Yaskawa INFORM job: R2_W27-A2(70,-90)_MP_OK.JBI

/JOB
//NAME R2_W27-A2(70,-90)_MP_OK
///FOLDERNAME MP_TEST
//POS
///NPOS 130,130,0,4,0,0
///TOOL 0
///POSTYPE PULSE
///PULSE
C00000=102318,51059,-6827,-6506,109190,54954
C00001=121032,58356,65608,-5376,86027,77236
C00002=120656,64598,75406,-5436,83192,77232
C00003=120505,64053,76314,-5460,82347,77219
C00004=120511,67645,82265,-5481,80539,77299
C00005=120505,64053,76314,-5460,82347,77219
C00006=120199,65070,76942,-5493,82463,77112
C00007=120032,61399,73230,-5508,82846,77040
C00008=120199,65070,76942,-5493,82463,77112
C00009=121567,62706,73730,-5333,83311,77530
C00010=121293,57658,68714,-5360,83784,77419
C00011=120253,58213,69266,-5476,83660,77079
C00012=121293,57658,68714,-5360,83784,77419
C00013=121567,62706,73730,-5333,83311,77530
C00014=120505,64053,76314,-5460,82347,77219
C00015=120656,64598,75406,-5436,83192,77232
C00016=121032,58526,65774,-5376,86013,77236
C00017=93357,59983,67350,2576,87301,77052
C00018=93973,65449,76277,2662,84599,77201
C00019=93950,64770,77022,2661,83793,77176
C00020=94041,68208,82724,2681,82050,77169
C00021=93950,64770,77022,2661,83793,77176
C00022=94821,64601,76206,2774,84179,77472
C00023=94634,60689,72295,2749,84583,77418
C00024=94821,64601,76206,2774,84179,77472
C00025=93392,64700,76725,2587,83958,76996
C00026=93160,58385,69524,2553,85150,76943
C00027=94147,57298,68173,2682,85392,77275
C00028=93160,58385,69524,2553,85150,76943
C00029=93392,64700,76725,2587,83958,76996
C00030=93950,64770,77022,2661,83793,77176
C00031=93973,65449,76277,2662,84599,77201
C00032=93336,59773,67146,2573,87319,77046
C00033=95545,69101,76731,-2374,84009,73270
C00034=95160,67852,79145,-2422,81872,73183
C00035=95003,67493,80298,-2443,80974,73148
C00036=94849,62700,75029,-2455,81748,73082
C00037=95003,67493,80298,-2443,80974,73148
C00038=93105,70422,84610,-2644,79768,72546
C00039=92524,67765,81382,-2700,80371,72342
C00040=93361,68913,82672,-2615,80194,72622
C00041=94751,59758,68035,-2453,84535,72995
C00042=92805,53349,62303,-2649,84709,72342
C00043=92901,55574,66096,-2644,83522,72399
C00044=92805,53349,62303,-2649,84709,72342
C00045=94751,59758,68035,-2453,84535,72995
C00046=95003,67493,80298,-2443,80974,73148
C00047=95160,67852,79145,-2422,81872,73183
C00048=95545,69101,76731,-2374,84009,73270
C00049=107317,62571,74358,10654,88778,76029
C00050=107317,56363,61014,10704,93717,76452
C00051=107317,62472,74242,10653,88798,76031
C00052=107230,62000,74261,10636,88556,75982
C00053=107581,65118,76915,10703,88484,76092
C00054=107323,60406,70480,10660,90030,76138
C00055=107264,61783,74050,10643,88577,75994
C00056=107253,61475,73709,10642,88626,75994
C00057=107117,62576,75125,9124,76631,64990
C00058=107127,63032,75625,10605,72549,55451
C00059=107164,62402,74962,9975,72602,48239
C00060=107192,61809,74312,8045,73320,42963
C00061=107223,63525,76074,7091,73334,41100
C00062=107292,63418,75963,5949,73527,39196
C00063=107230,61705,73943,5940,73892,39194
C00064=107323,62660,74463,4678,74173,37311
C00065=107324,62694,74502,4678,74166,37311
C00066=107665,73796,87925,4736,71600,37329
C00067=120729,48613,37887,-12949,101575,-14829
C00068=120728,62727,74542,-12584,86628,-80773
C00069=120664,61680,73824,-12594,86525,-80783
C00070=120693,60658,70774,-12585,87849,-80908
C00071=120585,65581,77469,-12610,86279,-80786
C00072=120690,61906,74287,-12590,86368,-80759
C00073=120903,61800,74113,-12557,86448,-80696
C00074=120945,62548,75100,-8817,74987,-69882
C00075=120948,62197,74655,-9458,70881,-60435
C00076=120932,61569,73990,-8829,71047,-53224
C00077=120988,63466,76076,-6164,72080,-46036
C00078=121112,63464,75917,-5072,72564,-44073
C00079=121088,62388,74845,-3850,73000,-42173
C00080=120728,62552,74336,-3837,73380,-42308
C00081=120720,61560,72154,180,93079,81636
C00082=120721,62738,74555,180,92207,81635
C00083=120791,87813,92293,81,108616,81679
C00084=120002,63379,75221,11,92127,81398
C00085=121441,63308,75123,350,92148,81873
C00086=120870,108608,123515,114,99903,81701
C00087=120721,62723,74537,180,92210,81635
C00088=120720,62741,74558,180,92206,81635
C00089=93952,63192,75095,14290,85903,-74473
C00090=93948,63106,74994,14289,85921,-74472
C00091=93949,63106,74994,14289,85921,-74472
C00092=93949,63106,74994,14289,85921,-74472
C00093=93511,61763,72320,14213,86923,-74505
C00094=94061,66569,78930,14314,85278,-74508
C00095=93933,62856,74699,14286,85975,-74471
C00096=93933,62856,74699,14286,85975,-74471
C00097=93932,62855,74699,14286,85976,-74471
C00098=93936,62941,74800,14287,85957,-74472
C00099=93954,63189,75092,-4074,77084,-70207
C00100=93950,63103,74990,-4074,77102,-70209
C00101=93950,63090,74975,-4074,77104,-70209
C00102=93949,63085,74969,-4074,77106,-70209
C00103=94045,66011,77989,-4076,76757,-70165
C00104=93880,61095,71289,-4060,78342,-70273
C00105=93963,63270,75188,-4074,77067,-70203
C00106=93963,63275,75194,-4074,77066,-70203
C00107=93963,63288,75209,-4074,77063,-70203
C00108=93967,63374,75311,-4074,77045,-70201
C00109=93937,63000,74869,-16709,69815,76001
C00110=93934,62914,74768,-16707,69832,75997
C00111=93932,62884,74733,-16706,69838,75996
C00112=93931,62873,74719,-16706,69840,75995
C00113=94312,65792,77997,-16780,69420,76194
C00114=94250,60204,70492,-16607,71084,75933
C00115=93941,62972,74836,-16709,69822,76001
C00116=93942,62984,74850,-16709,69819,76002
C00117=93943,63013,74885,-16710,69814,76003
C00118=93947,63099,74986,-16712,69797,76007
C00119=93938,62981,74847,-7114,69680,67691
C00120=93935,62895,74746,-7113,69698,67689
C00121=93933,62866,74712,-7113,69704,67688
C00122=93933,62855,74698,-7112,69706,67688
C00123=93919,60777,70917,-7059,70955,67609
C00124=94303,65238,77063,-7147,69509,67829
C00125=93920,62687,74500,-7110,69740,67681
C00126=93920,62698,74513,-7110,69738,67682
C00127=93922,62727,74547,-7111,69732,67682
C00128=93926,62812,74648,-7112,69715,67685
C00129=51349,-6233,-27963,187,103874,81653
BC00000=194563,177624,868736
BC00001=225604,138849,769169
BC00002=225604,138849,769169
BC00003=225604,138849,769169
BC00004=225604,138849,769169
BC00005=225604,138849,769169
BC00006=225604,138849,769169
BC00007=225604,138849,769169
BC00008=225604,138849,769169
BC00009=225604,138849,769169
BC00010=225604,138849,769169
BC00011=225604,138849,769169
BC00012=225604,138849,769169
BC00013=225604,138849,769169
BC00014=225604,138849,769169
BC00015=225604,138849,769169
BC00016=225604,138849,769169
BC00017=124341,124762,768464
BC00018=124341,124762,768464
BC00019=124341,124762,768464
BC00020=124341,124762,768464
BC00021=124341,124762,768464
BC00022=124341,124762,768464
BC00023=124341,124762,768464
BC00024=124341,124762,768464
BC00025=124341,124762,768464
BC00026=124341,124762,768464
BC00027=124341,124762,768464
BC00028=124341,124762,768464
BC00029=124341,124762,768464
BC00030=124341,124762,768464
BC00031=124341,124762,768464
BC00032=124341,124762,768464
BC00033=131551,156203,1070987
BC00034=131551,156203,1070987
BC00035=131551,156203,1070987
BC00036=131551,156203,1070987
BC00037=131551,156203,1070987
BC00038=131551,156203,1070987
BC00039=131551,156203,1070987
BC00040=131551,156203,1070987
BC00041=131551,156203,1070987
BC00042=131551,156203,1070987
BC00043=131551,156203,1070987
BC00044=131551,156203,1070987
BC00045=131551,156203,1070987
BC00046=131551,156203,1070987
BC00047=131551,156203,1070987
BC00048=131551,156203,1070987
BC00049=225137,131323,879040
BC00050=223667,125139,756323
BC00051=223667,125139,756323
BC00052=223075,126867,747658
BC00053=223075,126867,747658
BC00054=223075,126867,747658
BC00055=218396,127755,746641
BC00056=215210,128375,745961
BC00057=203609,151152,766146
BC00058=201855,161532,767450
BC00059=199281,163395,767937
BC00060=195364,163337,768565
BC00061=193166,166495,764643
BC00062=190579,170342,759829
BC00063=190579,170342,759829
BC00064=187290,170589,769799
BC00065=184872,170576,795413
BC00066=184861,181079,896469
BC00067=167411,129445,757678
BC00068=167411,129445,757678
BC00069=167997,131165,748991
BC00070=167997,131165,748991
BC00071=167997,131165,748991
BC00072=172685,131992,747792
BC00073=175877,132570,746989
BC00074=187923,154884,766916
BC00075=189976,165022,768336
BC00076=192744,166728,768846
BC00077=199094,169671,765390
BC00078=201778,173472,760485
BC00079=204162,173688,760124
BC00080=205164,173670,770332
BC00081=217813,145490,1075175
BC00082=217813,150433,1060626
BC00083=217813,152410,925547
BC00084=217813,152410,1052396
BC00085=217813,152410,1052396
BC00086=217813,152407,927156
BC00087=217772,148655,1043478
BC00088=217771,143712,1064054
BC00089=114600,133818,976434
BC00090=114611,123316,875378
BC00091=110715,126262,854320
BC00092=109157,127441,845897
BC00093=109157,127441,845897
BC00094=109157,127441,845897
BC00095=146537,130921,755729
BC00096=148095,129743,764153
BC00097=151990,126796,785211
BC00098=151980,137299,886266
BC00099=101051,138319,898903
BC00100=101062,127816,797847
BC00101=99318,130341,773149
BC00102=98620,131350,763270
BC00103=98620,131350,763270
BC00104=98620,131350,763270
BC00105=60690,124587,772909
BC00106=61388,123578,782788
BC00107=63132,121053,807486
BC00108=63122,131556,908542
BC00109=157999,142083,988332
BC00110=158010,131580,887276
BC00111=159966,134490,863290
BC00112=160748,135654,853695
BC00113=160748,135654,853695
BC00114=160748,135654,853695
BC00115=123117,139629,764979
BC00116=122335,138464,774574
BC00117=120379,135554,798560
BC00118=120368,146057,899616
BC00119=145080,148155,895629
BC00120=145090,137652,794573
BC00121=146786,140154,769808
BC00122=147464,141155,759903
BC00123=147464,141155,759903
BC00124=147464,141155,759903
BC00125=185325,133893,768075
BC00126=184646,132892,777981
BC00127=182951,130390,802745
BC00128=182941,140893,903801
BC00129=217772,217062,1064053
///POSTYPE BASE
///RECTAN
///RCONF 0,0,0,0,0,0,0,0,0,0,0,0,0,0,0,0,0,0,0,0,0,0,0,0
P00006=0.222,-3.123,-1.508,0.0000,0.0000,0.0000
P00011=-2.329,-0.061,-0.282,0.0000,0.0000,0.0000
P00012=-0.183,-1.308,1.069,0.0000,0.0000,0.0000
P00013=-0.119,0.591,-2.131,0.0000,0.0000,0.0000
//INST
///DATE 2023/11/16 10:47
///ATTR SC,RW
///GROUP1 RB1,BS1
NOP
'r2_W27-A2(70,-90)
'
'Path S829
SFTOF
MOVJ C00000 BC00000 VJ=20.00
MOVJ C00001 BC00001 VJ=20.00
MOVL C00002 BC00002 V=100.0
MOVL C00003 BC00003 V=60.0
REFP 3 C00004 BC00004
CALL JOB:SEARCH-R1
SET P011 P006
SFTON P011
MOVL C00005 BC00005 V=60.0
MOVL C00006 BC00006 V=60.0
REFP 3 C00007 BC00007
CALL JOB:SEARCH-R1
SET P011 P006
SFTON P011
MOVL C00008 BC00008 V=60.0
MOVL C00009 BC00009 V=100.0
MOVL C00010 BC00010 V=60.0
REFP 3 C00011 BC00011
CALL JOB:SEARCH-R1
SET P011 P006
SFTON P011
MOVL C00012 BC00012 V=60.0
MOVL C00013 BC00013 V=100.0
MOVL C00014 BC00014 V=100.0
MOVL C00015 BC00015 V=100.0
MOVL C00016 BC00016 V=100.0
'Path S830
SFTOF
MOVJ C00017 BC00017 VJ=20.00
MOVL C00018 BC00018 V=100.0
MOVL C00019 BC00019 V=60.0
REFP 3 C00020 BC00020
CALL JOB:SEARCH-R1
SET P012 P006
SFTON P012
MOVL C00021 BC00021 V=60.0
MOVL C00022 BC00022 V=60.0
REFP 3 C00023 BC00023
CALL JOB:SEARCH-R1
SET P012 P006
SFTON P012
MOVL C00024 BC00024 V=60.0
MOVL C00025 BC00025 V=100.0
MOVL C00026 BC00026 V=60.0
REFP 3 C00027 BC00027
CALL JOB:SEARCH-R1
SET P012 P006
SFTON P012
MOVL C00028 BC00028 V=60.0
MOVL C00029 BC00029 V=100.0
MOVL C00030 BC00030 V=100.0
MOVL C00031 BC00031 V=100.0
MOVL C00032 BC00032 V=100.0
'Path S831
SFTOF
MOVJ C00033 BC00033 VJ=20.00
MOVL C00034 BC00034 V=100.0
MOVL C00035 BC00035 V=60.0
REFP 3 C00036 BC00036
CALL JOB:SEARCH-R1
SET P013 P006
SFTON P013
MOVL C00037 BC00037 V=60.0
MOVL C00038 BC00038 V=60.0
REFP 3 C00039 BC00039
CALL JOB:SEARCH-R1
SET P013 P006
SFTON P013
MOVL C00040 BC00040 V=60.0
MOVL C00041 BC00041 V=100.0
MOVL C00042 BC00042 V=60.0
REFP 3 C00043 BC00043
CALL JOB:SEARCH-R1
SET P013 P006
SFTON P013
MOVL C00044 BC00044 V=60.0
MOVL C00045 BC00045 V=100.0
MOVL C00046 BC00046 V=100.0
MOVL C00047 BC00047 V=100.0
MOVL C00048 BC00048 V=1000.0
'Path W832
SFTOF
SFTON P011
MOVJ C00049 BC00049 VJ=20.00
MOVJ C00050 BC00050 VJ=20.00
MOVL C00051 BC00051 V=100.0
MOVL C00052 BC00052 V=100.0 PL=0
REFP 1 C00053 BC00053
REFP 2 C00054 BC00054
MACRO1 MJ#(0) ARGF7
ARCON
MOVL C00055 BC00055 V=10.0
MOVL C00056 BC00056 V=10.0
MOVL C00057 BC00057 V=11.7
MOVL C00058 BC00058 V=11.7
MOVL C00059 BC00059 V=11.7
MOVL C00060 BC00060 V=11.7
MOVL C00061 BC00061 V=10.0
MOVL C00062 BC00062 V=10.0
MOVL C00063 BC00063 V=10.0
ARCOF
MOVL C00064 BC00064 V=100.0
MOVL C00065 BC00065 V=100.0
SFTOF
MOVL C00066 BC00066 V=100.0
'Path VIA908
SFTOF
MOVJ C00067 BC00067 VJ=20.00
'Path W833
SFTOF
SFTON P012
MOVL C00068 BC00068 V=100.0
MOVL C00069 BC00069 V=100.0 PL=0
REFP 1 C00070 BC00070
REFP 2 C00071 BC00071
MACRO1 MJ#(0) ARGF7
ARCON
MOVL C00072 BC00072 V=10.0
MOVL C00073 BC00073 V=10.0
MOVL C00074 BC00074 V=13.3
MOVL C00075 BC00075 V=13.3
MOVL C00076 BC00076 V=13.3
MOVL C00077 BC00077 V=10.0
MOVL C00078 BC00078 V=10.0
MOVL C00079 BC00079 V=10.0
ARCOF
MOVL C00080 BC00080 V=100.0
SFTOF
'Path W834
SFTOF
SFTON P013
MOVJ C00081 BC00081 VJ=20.00
MOVL C00082 BC00082 V=100.0
MOVL C00083 BC00083 V=100.0 PL=0
REFP 1 C00084 BC00084
REFP 2 C00085 BC00085
MACRO1 MJ#(0) ARGF7
ARCON
MOVL C00086 BC00086 V=10.8
ARCOF
MOVL C00087 BC00087 V=100.0
MOVL C00088 BC00088 V=100.0
SFTOF
'BRAKUJACE BLASZKI
COMM 'Path W835
COMM SFTOF
COMM SFTON P012
COMM MOVJ C00089 BC00089 VJ=100.00
COMM MOVJ C00090 BC00090 VJ=100.00
COMM MOVL C00091 BC00091 V=400.0
COMM MOVL C00092 BC00092 V=100.0 PL=0
COMM REFP 1 C00093 BC00093
COMM REFP 2 C00094 BC00094
COMM MACRO1 MJ#(0) ARGF0
COMM ARCON
COMM MOVL C00095 BC00095 V=10.0
COMM ARCOF
COMM MOVL C00096 BC00096 V=400.0
COMM MOVL C00097 BC00097 V=1000.0
COMM MOVL C00098 BC00098 V=1000.0
COMM SFTOF
COMM 'Path W836
COMM SFTOF
COMM SFTON P012
COMM MOVJ C00099 BC00099 VJ=100.00
COMM MOVJ C00100 BC00100 VJ=100.00
COMM MOVL C00101 BC00101 V=400.0
COMM MOVL C00102 BC00102 V=100.0 PL=0
COMM REFP 1 C00103 BC00103
COMM REFP 2 C00104 BC00104
COMM MACRO1 MJ#(0) ARGF0
COMM ARCON
COMM MOVL C00105 BC00105 V=10.0
COMM ARCOF
COMM MOVL C00106 BC00106 V=400.0
COMM MOVL C00107 BC00107 V=1000.0
COMM MOVL C00108 BC00108 V=1000.0
COMM SFTOF
COMM 'Path W837
COMM SFTOF
COMM SFTON P011
COMM MOVJ C00109 BC00109 VJ=100.00
COMM MOVJ C00110 BC00110 VJ=100.00
COMM MOVL C00111 BC00111 V=400.0
COMM MOVL C00112 BC00112 V=100.0 PL=0
COMM REFP 1 C00113 BC00113
COMM REFP 2 C00114 BC00114
COMM MACRO1 MJ#(0) ARGF0
COMM ARCON
COMM MOVL C00115 BC00115 V=10.0
COMM ARCOF
COMM MOVL C00116 BC00116 V=400.0
COMM MOVL C00117 BC00117 V=1000.0
COMM MOVL C00118 BC00118 V=1000.0
COMM SFTOF
COMM 'Path W838
COMM SFTOF
COMM SFTON P011
COMM MOVJ C00119 BC00119 VJ=100.00
COMM MOVJ C00120 BC00120 VJ=100.00
COMM MOVL C00121 BC00121 V=400.0
COMM MOVL C00122 BC00122 V=100.0 PL=0
COMM REFP 1 C00123 BC00123
COMM REFP 2 C00124 BC00124
COMM MACRO1 MJ#(0) ARGF0
COMM ARCON
COMM MOVL C00125 BC00125 V=10.0
COMM ARCOF
COMM MOVL C00126 BC00126 V=400.0
COMM MOVL C00127 BC00127 V=1000.0
COMM MOVL C00128 BC00128 V=1000.0
COMM SFTOF
MOVJ C00129 BC00129 VJ=20.00
END
